// Mitsubishi GX Works2 project: TestData01   PLC: Q13UDV

PROGRAM MAIN
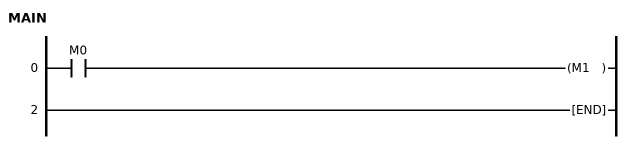
0     LD      M0
      OUT     M1
2     END
END_PROGRAM
